// TwinCAT 3 PLC project TEST
// ProgramVersion: 3.1.4023.0
// libraries:
//   Tc2_BABasic, * (Beckhoff Automation GmbH)
//   Tc2_Standard, * (Beckhoff Automation GmbH)
//   Tc2_System, * (Beckhoff Automation GmbH)
//   Tc3_Module, * (Beckhoff Automation GmbH)
// project tree:
//   / GlobalTextList.TcGTLO, PlcTask.TcTTO, Visualization Manager.TcVMO (not stored)
//   POUs/ MAIN.TcPOU
//   VISUs/ Visualization.TcVIS

CONFIGURATION TEST
    RESOURCE PLC ON TwinCAT3
        TASK PlcTask(INTERVAL := T#10ms, PRIORITY := 22);
        PROGRAM MAIN WITH PlcTask : MAIN;
    END_RESOURCE
END_CONFIGURATION

// ---- POUs/MAIN.TcPOU
PROGRAM MAIN

VAR_INPUT
	SWITCH : BOOL;
END_VAR

VAR_OUTPUT
	LED : BOOL;
END_VAR

VAR
	FB_SingleDoubleClick : FB_SingleDoubleClick; 
END_VAR

FB_SingleDoubleClick(bSwitch:= SWITCH, tSwitchTime:= T#500MS);

IF FB_SingleDoubleClick.bSingleClick THEN
	LED := TRUE;
	SWITCH := FALSE;

END_IF

END_PROGRAM

// ---- VISUs/Visualization.TcVIS
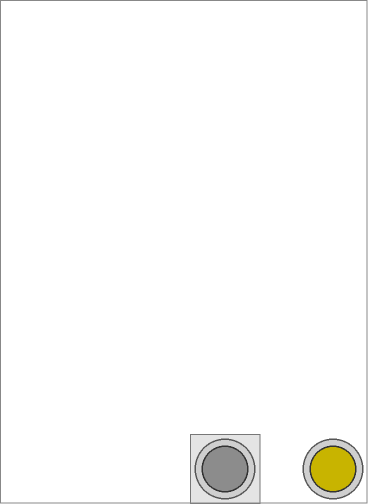
VISUALIZATION Visualization  // 368x504
    PushSwitch (190,434 70x70), variable: MAIN.SWITCH, behaviour: TOGGLE, style: Switch-PushSwitch-Gray
    Lamp1 (298,434 70x70), variable: MAIN.LED, style: Lamp-Lamp1-Yellow
END_VISUALIZATION
